// TIA Portal V21 export
VAR_GLOBAL   // PLC tag table "K_Tema"
END_VAR
VAR_GLOBAL CONSTANT   // user constants
   K_Tema_StdDubit : Int := 0;
   K_Tema_StdBrain : Int := 1;
END_VAR
